(* IEC 61131-3 sources: repolevel_ST_code_completion/real_groud_truth最新/repoeval_readwriteFile/readful_result, 2 files *)

(* ---- ReadFile.st ---- *)
VAR
	nState	:	BYTE;
	fileHandle	:	UDINT;//文件句柄
	readBuffer	:	ARRAY[0..255] OF BYTE;//读取数据缓冲区
	nNumRead	:	UDINT;//读取文件的字节数
	fbRtrig	:	R_TRIG;//实例化上升沿触发功能块
END_VAR
VAR_OUTPUT
	bDone	:	BOOL;//读取成功
	bBusy	:	BOOL;//读取忙
	bErr	:	BOOL;//读取出错
	nErrId	:	UDINT;//错误代码
	readData	:	ARRAY[0..255] OF BYTE;//读取的数据
END_VAR

CASE nState OF
	0:
		fbRtrig(CLK := bExec);//等待用户触发调用
		IF fbRtrig.Q THEN
			nState := 1;
			bBusy := TRUE;
			bErr := FALSE;
			nErrId := 0;
			bDone := FALSE;
		END_IF;

	1:
		// 打开文件
		fileHandle := FileOpen(fileName := fileName, mode := 'READ');
		IF fileHandle = 0 THEN
			bErr := TRUE;
			nErrId := 1; // 文件打开失败
			nState := 0;
			bBusy := FALSE;
		ELSE
			nState := 2;
		END_IF;

	2:
		// 读取文件内容
		nNumRead := FileRead(fileHandle := fileHandle, buffer := readBuffer, size := SIZEOF(readBuffer));
		IF nNumRead = 0 THEN
			bErr := TRUE;
			nErrId := 2; // 文件读取失败
			nState := 0;
			bBusy := FALSE;
		ELSE
			readData := readBuffer; // 将读取的数据存储到输出变量
			nState := 3;
		END_IF;

	3:
		// 关闭文件
		IF FileClose(fileHandle := fileHandle) THEN
			bDone := TRUE;
			bBusy := FALSE;
			nState := 0;
		ELSE
			bErr := TRUE;
			nErrId := 3; // 文件关闭失败
			nState := 0;
			bBusy := FALSE;
		END_IF;

ELSE
	nState := 0;
END_CASE;

(* ---- WriteFile.st ---- *)
VAR
	nState	:	BYTE;
	fileHandle	:	UDINT;//文件句柄
	i	:	BYTE;//定义循环变量

	fbRtrig	:	R_TRIG;//实例化上升沿触发功能块
END_VAR
VAR_OUTPUT
	bDone	:	BOOL;//写入成功
	bBusy	:	BOOL;//写入忙
	bErr	:	BOOL;//写入出错
	nErrId	:	UDINT;//错误代码
END_VAR

CASE nState OF
	0:
		fbRtrig(CLK := bExec);//等待用户触发调用
		IF fbRtrig.Q THEN
			nState := 1;
			bBusy := TRUE;
			bErr := FALSE;
			nErrId := 0;
			bDone := FALSE;
		END_IF
	1:
		// 打开文件
		fileHandle := SysFileOpen(szFile := fileName, am := 'w');//以写模式打开文件
		IF fileHandle = 0 THEN
			nState := 99; // 错误状态
			bErr := TRUE;
			nErrId := 1; // 文件打开失败
		ELSE
			nState := 2;
		END_IF
	2:
		// 写入文件
		IF SysFileWrite(hFile := fileHandle, pBuffer := ADR(writeBuffer), szSize := writeNum) THEN
			nState := 3;
		ELSE
			nState := 99; // 错误状态
			bErr := TRUE;
			nErrId := 2; // 写入失败
		END_IF
	3:
		// 关闭文件
		IF SysFileClose(hFile := fileHandle) THEN
			nState := 4;
		ELSE
			nState := 99; // 错误状态
			bErr := TRUE;
			nErrId := 3; // 文件关闭失败
		END_IF
	4:
		// 写入完成
		bDone := TRUE;
		bBusy := FALSE;
		nState := 0; // 重置状态
	99:
		// 错误处理
		bBusy := FALSE;
	END_CASE
END_FUNCTION_BLOCK
